SYSTEM VDMA_V3
  (* Version 1.0, 2025-04-16, DEVIASH *)
  APPLICATION VDMA_V3App
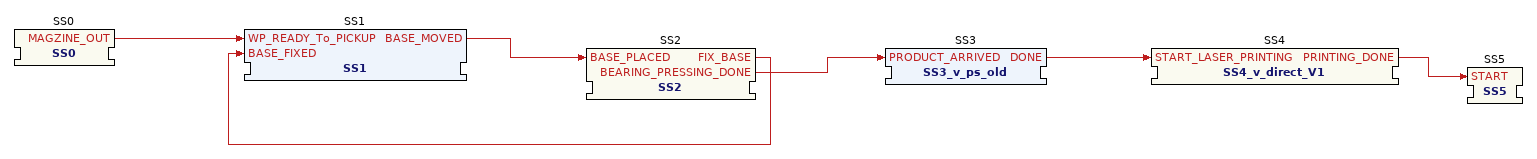
    FBS
      SS0 : SS0;
      SS2 : SS2;
      SS4 : UserLibs::SubStations::SS4::SS4_v_direct_V1;
      SS5 : UserLibs::SubStations::SS5::SS5;
    END_FBS
    SUBAPPS
      SS1 : SS1;
      SS3 : SS3_v_ps_old;
    END_SUBAPPS
    EVENT_CONNECTIONS
      SS0.MAGZINE_OUT TO SS1.WP_READY_To_PICKUP;
      SS1.BASE_MOVED TO SS2.BASE_PLACED;
      SS2.FIX_BASE TO SS1.BASE_FIXED;
      SS2.BEARING_PRESSING_DONE TO SS3.PRODUCT_ARRIVED;
      SS3.DONE TO SS4.START_LASER_PRINTING;
      SS4.PRINTING_DONE TO SS5.START;
    END_CONNECTIONS
  END_APPLICATION
  DEVICE FORTE_PC : FORTE_PC(MGR_ID := "localhost:61499" (* Device manager socket ID *))
    {SET_ATTRIBUTE(Profile, HOLOBLOC)}
    RESOURCE EMB_RES : EMB_RES
    END_RESOURCE
  END_DEVICE
END_SYSTEM
